% RSLogix 500 project PARKING GARAGE_BAK003.RSS, saved by version 8.30.00.16 %
PROJECT "UNTITLED"    % processor: MicroLogix 1000 %

PROGRAM FILES
  LAD 2 "MAIN_PROG"  8 rungs
  LAD 3 "USER_FAULT"  1 rungs
  LAD 4 "HSC_INT"  1 rungs
  LAD 5 "STI_INT"  1 rungs
  LAD 6, 7, 8, 9, 10, 11, 12, 13, 14, 15, 16: only END

DATA FILES
  O0 OUTPUT  1 elements
  I1 INPUT  2 elements
  S2 STATUS  33 elements
  B3 BINARY  32 elements
  T4 TIMER  40 elements
  C5 COUNTER  32 elements
  R6 CONTROL  16 elements
  N7 INTEGER  105 elements

LADDER 2 "MAIN_PROG"
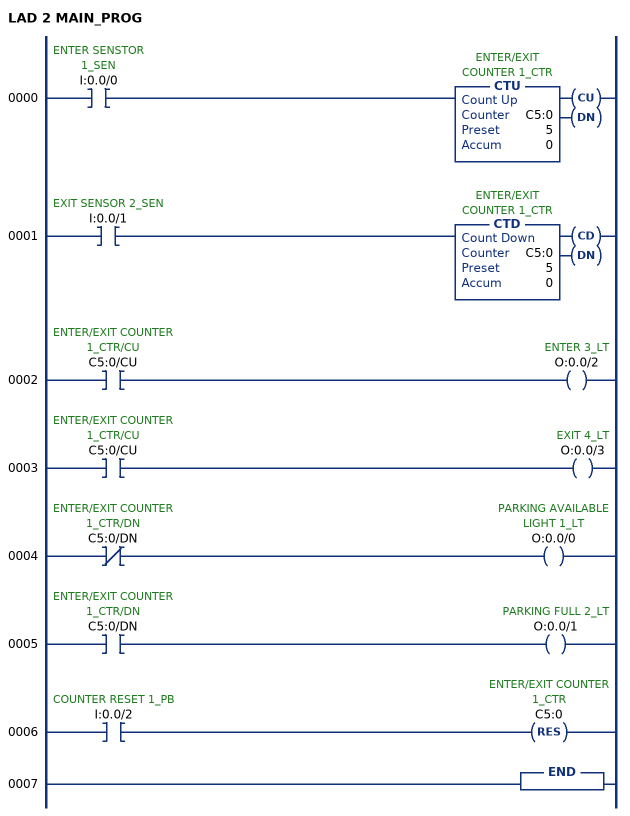
% Rung: 0 %
SOR XIC I:0.0/0 CTU C5:0 5 0 EOR
%   I:0.0/0  1_SEN  "ENTER SENSTOR" %
%   C5:0  1_CTR  "ENTER/EXIT COUNTER" %
% Rung: 1 %
SOR XIC I:0.0/1 CTD C5:0 5 0 EOR
%   I:0.0/1  2_SEN  "EXIT SENSOR" %
%   C5:0  1_CTR  "ENTER/EXIT COUNTER" %
% Rung: 2 %
SOR XIC C5:0/CU OTE O:0.0/2 EOR
%   C5:0  1_CTR  "ENTER/EXIT COUNTER" %
%   O:0.0/2  3_LT  "ENTER" %
% Rung: 3 %
SOR XIC C5:0/CU OTE O:0.0/3 EOR
%   C5:0  1_CTR  "ENTER/EXIT COUNTER" %
%   O:0.0/3  4_LT  "EXIT" %
% Rung: 4 %
SOR XIO C5:0/DN OTE O:0.0/0 EOR
%   C5:0  1_CTR  "ENTER/EXIT COUNTER" %
%   O:0.0/0  1_LT  "PARKING AVAILABLE LIGHT" %
% Rung: 5 %
SOR XIC C5:0/DN OTE O:0.0/1 EOR
%   C5:0  1_CTR  "ENTER/EXIT COUNTER" %
%   O:0.0/1  2_LT  "PARKING FULL" %
% Rung: 6 %
SOR XIC I:0.0/2 RES C5:0 EOR
%   I:0.0/2  1_PB  "COUNTER RESET" %
%   C5:0  1_CTR  "ENTER/EXIT COUNTER" %
% Rung: 7 %
SOR END EOR

DATA TABLE (non-zero values as saved)
DATA C5
% .PRE .ACC %
% C5:0 % 5 0
